INTERFACE I_HE_SATT_FilterToTransmission


METHOD PUBLIC CalculateTransmission
VAR_INPUT
    fPhotonEnergy_eV : LREAL;
    iFilter : I_HE_SATT_Filter;
END_VAR
VAR_OUTPUT
    fMinimumTransmission : LREAL;
    fMaximumTransmission : LREAL;
END_VAR
END_METHOD

END_INTERFACE

(* stored: Version 1.1.0.1
   Itf I_HE_SATT_FilterToTransmission: Id {9f20e632-f820-449e-813d-b3cd6cce596a}
   Method CalculateTransmission: Id {3eec553f-a66d-4eb0-bdf8-aa9baadd974c} *)
